(* PLC project  *)

CONFIGURATION Empty_Module_24
END_CONFIGURATION
